// Mitsubishi GX Works2 project: SKUBI_program_worked   PLC: FX1N/FX1NC

PROGRAM MAIN
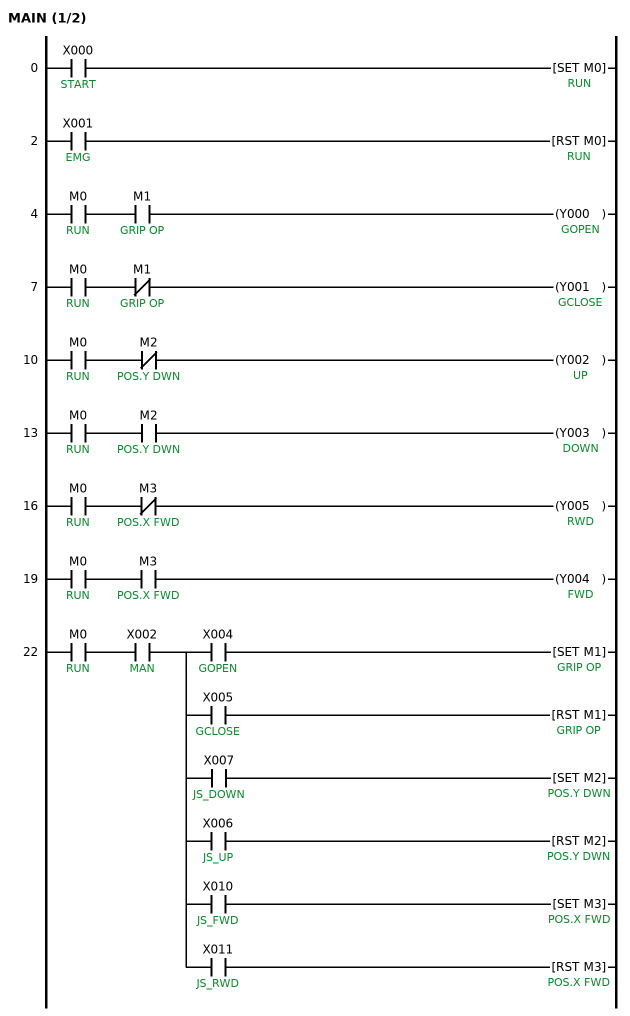
0     LD      X000  ; START
      SET     M0  ; RUN
2     LD      X001  ; EMG
      RST     M0  ; RUN
4     LD      M0  ; RUN
      AND     M1  ; GRIP OP
      OUT     Y000  ; GOPEN
7     LD      M0  ; RUN
      ANI     M1  ; GRIP OP
      OUT     Y001  ; GCLOSE
10    LD      M0  ; RUN
      ANI     M2  ; POS.Y DWN
      OUT     Y002  ; UP
13    LD      M0  ; RUN
      AND     M2  ; POS.Y DWN
      OUT     Y003  ; DOWN
16    LD      M0  ; RUN
      ANI     M3  ; POS.X FWD
      OUT     Y005  ; RWD
19    LD      M0  ; RUN
      AND     M3  ; POS.X FWD
      OUT     Y004  ; FWD
22    LD      M0  ; RUN
      AND     X002  ; MAN
      MPS
      AND     X004  ; GOPEN
      SET     M1  ; GRIP OP
      MRD
      AND     X005  ; GCLOSE
      RST     M1  ; GRIP OP
      MRD
      AND     X007  ; JS_DOWN
      SET     M2  ; POS.Y DWN
      MRD
      AND     X006  ; JS_UP
      RST     M2  ; POS.Y DWN
      MRD
      AND     X010  ; JS_FWD
      SET     M3  ; POS.X FWD
      MPP
      AND     X011  ; JS_RWD
      RST     M3  ; POS.X FWD
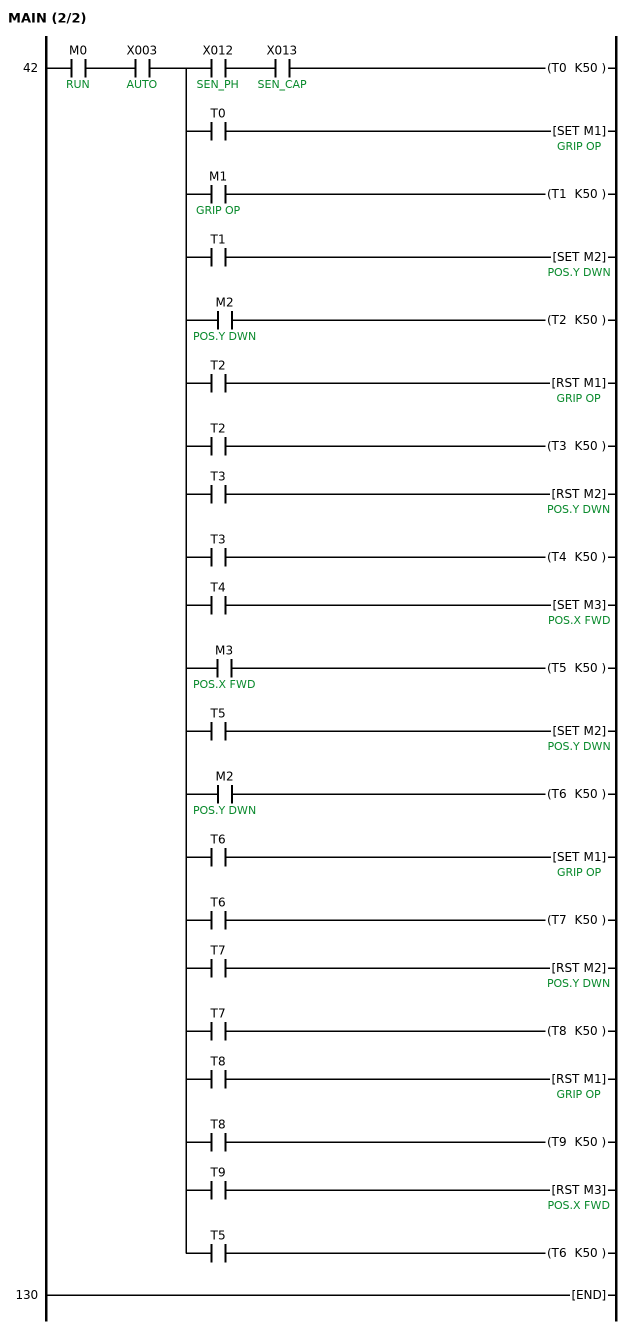
42    LD      M0  ; RUN
      AND     X003  ; AUTO
      MPS
      AND     X012  ; SEN_PH
      AND     X013  ; SEN_CAP
      OUT     T0 K50
      MRD
      AND     T0
      SET     M1  ; GRIP OP
      MRD
      AND     M1  ; GRIP OP
      OUT     T1 K50
      MRD
      AND     T1
      SET     M2  ; POS.Y DWN
      MRD
      AND     M2  ; POS.Y DWN
      OUT     T2 K50
      MRD
      AND     T2
      RST     M1  ; GRIP OP
      MRD
      AND     T2
      OUT     T3 K50
      MRD
      AND     T3
      RST     M2  ; POS.Y DWN
      MRD
      AND     T3
      OUT     T4 K50
      MRD
      AND     T4
      SET     M3  ; POS.X FWD
      MRD
      AND     M3  ; POS.X FWD
      OUT     T5 K50
      MRD
      AND     T5
      SET     M2  ; POS.Y DWN
      MRD
      AND     M2  ; POS.Y DWN
      OUT     T6 K50
      MRD
      AND     T6
      SET     M1  ; GRIP OP
      MRD
      AND     T6
      OUT     T7 K50
      MRD
      AND     T7
      RST     M2  ; POS.Y DWN
      MRD
      AND     T7
      OUT     T8 K50
      MRD
      AND     T8
      RST     M1  ; GRIP OP
      MRD
      AND     T8
      OUT     T9 K50
      MRD
      AND     T9
      RST     M3  ; POS.X FWD
      MPP
      AND     T5
      OUT     T6 K50
130   END
END_PROGRAM
